PROGRAM MAIN
VAR
	Hough: Hough;
	
END_VAR

Hough();

END_PROGRAM

(* stored: Version 1.1.0.1, ProductVersion 3.1.4024.12
   POU MAIN: Id {3832b137-74f0-4fa9-af16-a60b81154585}, SpecialFunc None *)
